// TIA Portal project "ACTEA_Ex5_ap" (V15.1)

(* hardware
DEVICE "S7-1200 station_2"  S7-1200 Station
   slot 0: "Rack_0"  S7-1200 Rack  Rack  V1.0
   slot 1: "PLC_1"  CPU 1215C DC/DC/Rly  6ES7 215-1HG31-0XB0  V3.0
*)

// ===== PLC "PLC_1"  CPU 1215C DC/DC/Rly =====

VAR_GLOBAL   // PLC tag table "Default tag table"
   "System_Byte" AT %MB254 : Byte;
   "FirstScan" AT %M254.0 : Bool;
   "DiagStatusUpdate" AT %M254.1 : Bool;
   "AlwaysTRUE" AT %M254.2 : Bool;
   "AlwaysFALSE" AT %M254.3 : Bool;
   "Clock_Byte" AT %MB255 : Byte;
   "Clock_10Hz" AT %M255.0 : Bool;
   "Clock_5Hz" AT %M255.1 : Bool;
   "Clock_2.5Hz" AT %M255.2 : Bool;
   "Clock_2Hz" AT %M255.3 : Bool;
   "Clock_1.25Hz" AT %M255.4 : Bool;
   "Clock_1Hz" AT %M255.5 : Bool;
   "Clock_0.625Hz" AT %M255.6 : Bool;
   "Clock_0.5Hz" AT %M255.7 : Bool;
   "iCC_BtnStop_S1" AT %I0.0 : Bool;   // Stop Button
   "iCC_BtnStartFw_S3" AT %I0.2 : Bool;   // Start button forward
   "iCC_McbMot_QM1" AT %I1.1 : Bool;   // Motor circuit breaker
   "iCC_ConMotFw_KM1" AT %I1.2 : Bool;   // Feedback signal contactor forward
   "oCC_LmpStartFw_H1" AT %Q0.0 : Bool;   // Lamp start forward
   "oCC_LmpStop_H3" AT %Q0.2 : Bool;   // Lamp stop
   "oCC_ConMotFw_KM1" AT %Q0.6 : Bool;   // Contactor motor forward
   "mMotStartedFw" AT %M0.0 : Bool;   // Motor started forward
   "iCC_SwiDolDor_S4" AT %I0.4 : Bool;   // Selection switch DOL DOR
   "iCC_BtnStartBw_S4" AT %I0.3 : Bool;   // Start button Backward
   "iCC_ConMotBw_KM2" AT %I1.4 : Bool;   // Feedback signal contactor backward
   "oCC_LmpStartBw_H2" AT %Q0.1 : Bool;   // Lamp start backward
   "oCC_ConMotBw_KM2" AT %Q0.7 : Bool;   // Contactor motor backward
   "mMotStartedBw" AT %M0.1 : Bool;   // Motor started backward
END_VAR

FUNCTION "FC_DOL" : Void   // FC1, FBD
{ S7_Optimized_Access := 'TRUE' }
VERSION : 0.1
BEGIN

REGION Network 1: Start-stop circuit "mMotStarted"
   // Start circuit = Start button
   // Stop circuit = Stop button AND Motor circuit breaker
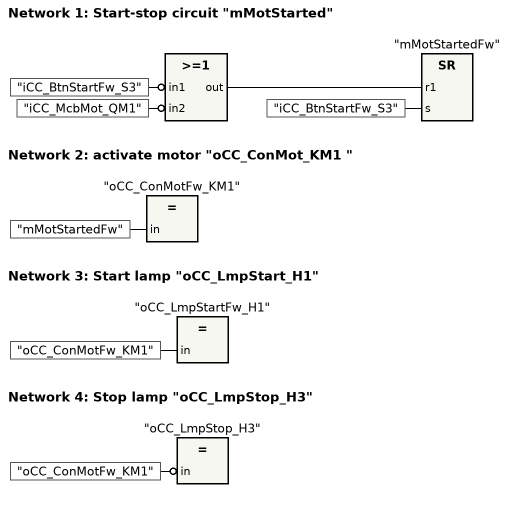
   IF "iCC_BtnStartFw_S3" THEN
       "mMotStartedFw" := TRUE;   // SR flip-flop
   END_IF;
   IF NOT "iCC_BtnStartFw_S3" OR NOT "iCC_McbMot_QM1" THEN "mMotStartedFw" := FALSE; END_IF;
END_REGION

REGION Network 2: activate motor "oCC_ConMot_KM1 "
   // Motor activation
   "oCC_ConMotFw_KM1" := "mMotStartedFw";
END_REGION

REGION Network 3: Start lamp "oCC_LmpStart_H1"
   // contactor feedback signal to (de)activate the lamp
   "oCC_LmpStartFw_H1" := "oCC_ConMotFw_KM1";
END_REGION

REGION Network 4: Stop lamp "oCC_LmpStop_H3"
   // contactor feedback signal to (de)activate the lamp
   "oCC_LmpStop_H3" := NOT "oCC_ConMotFw_KM1";
END_REGION
END_FUNCTION

FUNCTION "FC_DOR" : Void   // FC2, FBD
{ S7_Optimized_Access := 'TRUE' }
VERSION : 0.1
BEGIN

REGION Network 1: Start-stop circuit forward "mMotStartedFw"
   // Start circuit = Start button forward AND NOT backward started
   // Stop circuit = Stop button AND Motor circuit breaker
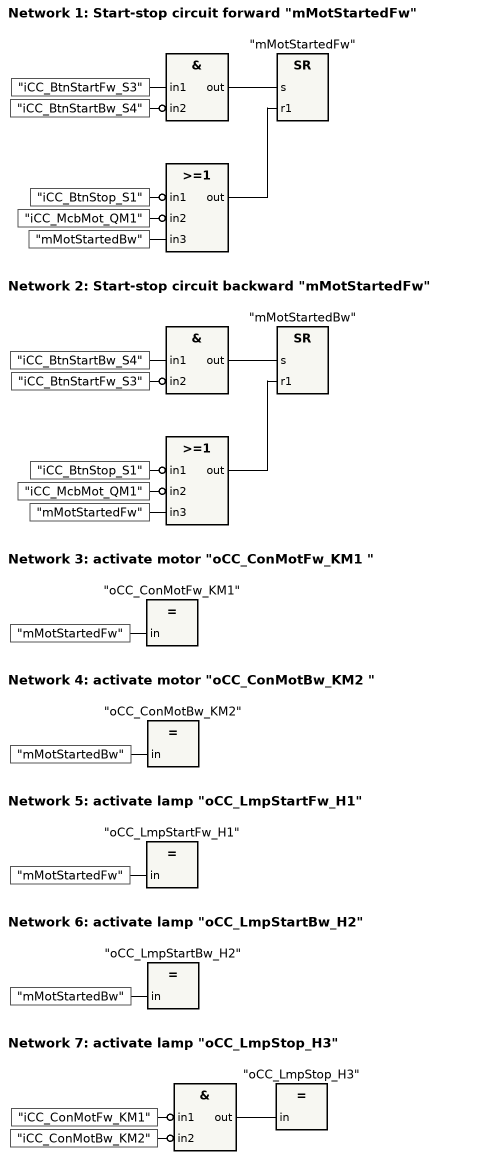
   IF "iCC_BtnStartFw_S3" AND NOT "iCC_BtnStartBw_S4" THEN
       "mMotStartedFw" := TRUE;   // SR flip-flop
   END_IF;
   IF NOT "iCC_BtnStop_S1" OR NOT "iCC_McbMot_QM1" OR "mMotStartedBw" THEN "mMotStartedFw" := FALSE; END_IF;
END_REGION

REGION Network 2: Start-stop circuit backward "mMotStartedFw"
   // Start circuit = Start button backward AND NOT forward started
   // Stop circuit = Stop button AND Motor circuit breaker
   IF "iCC_BtnStartBw_S4" AND NOT "iCC_BtnStartFw_S3" THEN
       "mMotStartedBw" := TRUE;   // SR flip-flop
   END_IF;
   IF NOT "iCC_BtnStop_S1" OR NOT "iCC_McbMot_QM1" OR "mMotStartedFw" THEN "mMotStartedBw" := FALSE; END_IF;
END_REGION

REGION Network 3: activate motor "oCC_ConMotFw_KM1 "
   // Motor activation
   "oCC_ConMotFw_KM1" := "mMotStartedFw";
END_REGION

REGION Network 4: activate motor "oCC_ConMotBw_KM2 "
   // Motor activation
   "oCC_ConMotBw_KM2" := "mMotStartedBw";
END_REGION

REGION Network 5: activate lamp "oCC_LmpStartFw_H1"
   // Control lamp green forward
   "oCC_LmpStartFw_H1" := "mMotStartedFw";
END_REGION

REGION Network 6: activate lamp "oCC_LmpStartBw_H2"
   // Control lamp green backward
   "oCC_LmpStartBw_H2" := "mMotStartedBw";
END_REGION

REGION Network 7: activate lamp "oCC_LmpStop_H3"
   // Control lamp red
   "oCC_LmpStop_H3" := NOT "iCC_ConMotFw_KM1" AND NOT "iCC_ConMotBw_KM2";
END_REGION
END_FUNCTION

ORGANIZATION_BLOCK "Main"   // OB1, LAD, ProgramCycle
TITLE = "Main Program Sweep (Cycle)"
{ S7_Optimized_Access := 'TRUE' }
VERSION : 0.1
BEGIN

REGION Network 1
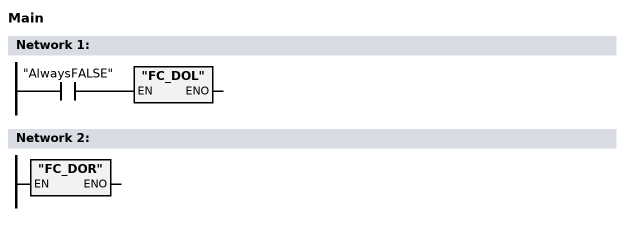
   RUNG wire#powerrail
      Contact( "AlwaysFALSE" )
      "FC_DOL"()
   END_RUNG
   // the same network as SCL:
   IF "AlwaysFALSE" THEN "FC_DOL"(); END_IF;
END_REGION

REGION Network 2
   RUNG wire#powerrail
      "FC_DOR"()
   END_RUNG
   // the same network as SCL:
   "FC_DOR"();
END_REGION
END_ORGANIZATION_BLOCK